PROGRAM PRG_FB_DigitalOutput_Test
VAR
	bFirstCycle		: BOOL := TRUE;
	bValue			: BOOL;					(* Output value to set on object *)
	poTestOutput	: FB_DigitalOutput();	(* Digital output object *)
END_VAR

IF bFirstCycle THEN
	bFirstCycle := FALSE;
	poTestOutput.MR_FirstCycle('My test digital output');
END_IF

poTestOutput.Out := bValue;
poTestOutput();

END_PROGRAM

(* stored: Version 1.1.0.1, ProductVersion 3.1.4024.9
   POU PRG_FB_DigitalOutput_Test: Id {ab5f3dff-b5ad-464c-933e-27a9747ff628}, SpecialFunc None *)
